//---------------------------------------------------------------------------------------------------------------
//
//  HAUD 2026.03.21
//
//  - MAIN_APPLICATION helper
//    - example PRG for setting up your application startup
//
//---------------------------------------------------------------------------------------------------------------
// This SOFTWARE is provided as an Example by THE PROVIDER "as is" and "with all faults." THE PROVIDER makes no 
// representations or warranties of any kind concerning the safety, suitability, lack of viruses, inaccuracies, 
// typographical errors, or other harmful components of this SOFTWARE. There are inherent dangers in the use of 
// any software, and you are solely responsible for determining whether this SOFTWARE is compatible with your 
// equipment and other software installed on your equipment. You are also solely responsible for the protection 
// of your equipment and backup of your data, and THE PROVIDER will not be liable for any damages you may suffer 
// in connection with using, modifying, or distributing this SOFTWARE.
//---------------------------------------------------------------------------------------------------------------
PROGRAM MAIN_APP
VAR
  eInit      AT %Q*     : E_PROGRESS;   // startup state machine after MAIN is initialized
  bXmlStartup           : BOOL;         // optional example switch for using xml configuration

  rDefaultJerk          : REAL := 400_000.0;
  rDefaultAccDec        : REAL :=  12_500.0;
  rDefaultVeloMax       : REAL :=   3_000.0;
  rDefaultVeloMin       : REAL :=   1_500.0;
  rDefaultGap           : REAL :=      76.0;
END_VAR

//-----------------------------------------------------------------------------
// check mapping switch
//-----------------------------------------------------------------------------
IF NOT MAPPING_in.BypassSwitch 
THEN 
  //eInit                                       := E_PROGRESS.PROGRESS_NOT_EXIST; 
END_IF
//-----------------------------------------------------------------------------
// wait for initialization to be complete before work may start
//-----------------------------------------------------------------------------
IF NOT (Main.eInit = E_PROGRESS.PROGRESS_DONE)
THEN
  eInit                                       := E_PROGRESS.PROGRESS_INIT;
  RETURN;
END_IF
//-----------------------------------------------------------------------------
//-----------------------------------------------------------------------------
// start your application init from here (example)
//-----------------------------------------------------------------------------
CASE eInit
OF
  //---------------------------------------------------------------------------
  E_PROGRESS.PROGRESS_NOT_EXIST:
    RETURN;       // you just bypassed the mapping
                  // check if you require anything from the initialisation
  //---------------------------------------------------------------------------
  E_PROGRESS.PROGRESS_INIT:
    GVL_APPLICATION.ConfigCtrl.Cmd            := E_DATA_CTRL.NULL;
    eInit                                     := E_PROGRESS.PROGRESS_BUSY;

  //---------------------------------------------------------------------------
  E_PROGRESS.PROGRESS_BUSY:
    IF NOT bXmlStartup
    THEN
      StationParameterExample();
      eInit                                   := E_PROGRESS.PROGRESS_WORKING;
    ELSE
      GVL_APPLICATION.ConfigCtrl.Cmd          := E_DATA_CTRL.INIT;
      eInit                                   := E_PROGRESS.PROGRESS_PREPARE;
    END_IF

  //---------------------------------------------------------------------------
  E_PROGRESS.PROGRESS_PREPARE:
    IF (GVL_APPLICATION.ConfigState.State = E_DATA_STATE.INIT + E_PROGRESS.PROGRESS_DONE)
    THEN
      GVL_APPLICATION.ConfigCtrl.Cmd          := E_DATA_CTRL.READ;
      eInit                                   := E_PROGRESS.PROGRESS_STARTUP;
    END_IF

  E_PROGRESS.PROGRESS_STARTUP:
    IF (GVL_APPLICATION.ConfigState.State = E_DATA_STATE.READ + E_PROGRESS.PROGRESS_DONE)
    THEN
      GVL_APPLICATION.ConfigCtrl.Cmd          := E_DATA_CTRL.NULL;
      eInit                                   := E_PROGRESS.PROGRESS_CHECK;
    END_IF

  E_PROGRESS.PROGRESS_CHECK:
    eInit                                     := E_PROGRESS.PROGRESS_OCCUPIED;

  E_PROGRESS.PROGRESS_OCCUPIED:
    eInit                                     := E_PROGRESS.PROGRESS_WORKING;

  E_PROGRESS.PROGRESS_WORKING:
    eInit                                     := E_PROGRESS.PROGRESS_DONE;
END_CASE
//-----------------------------------------------------------------------------
//-----------------------------------------------------------------------------
//-----------------------------------------------------------------------------
// connect data and control to xml configuration
GVL_APPLICATION.StationConfig.Identity        :=   GVL_XTS.Xpu.XpuOtcid;
GVL_APPLICATION.StationConfig.Ctrl            REF= GVL_APPLICATION.ConfigCtrl;
GVL_APPLICATION.StationConfig.State           REF= GVL_APPLICATION.ConfigState;

GVL_APPLICATION.StationConfig.MessageDevice   := e_Device.Device_Configuration;
GVL_APPLICATION.StationConfig.MessageLevel    := GVL_MSG.MessageLevel;
GVL_APPLICATION.StationConfig.FolderPath      := GVL_MSG.CON_DIR;
GVL_APPLICATION.StationConfig.StationParameter:= ADR(GVL_XTS.StationParameter);

GVL_APPLICATION.StationConfig();        // call xml configuration
//-----------------------------------------------------------------------------
//-----------------------------------------------------------------------------

END_PROGRAM

(* stored: Version 1.1.0.1, ProductVersion 3.1.4026.18
   POU MAIN_APP: Id {589cd8b7-b619-4bed-ad7a-c17614b60e90}, SpecialFunc None *)
